Fanuc TP program (LS listing): message22.ls

/PROG  MESSAGE22	  Macro
/ATTR
OWNER		= MNEDITOR;
COMMENT		= "USER MESSAGE";
PROG_SIZE	= 279;
CREATE		= DATE 22-05-23  TIME 16:17:10;
MODIFIED	= DATE 22-05-23  TIME 16:26:38;
FILE_NAME	= MESSAGE2;
VERSION		= 0;
LINE_COUNT	= 3;
MEMORY_SIZE	= 655;
PROTECT		= READ_WRITE;
TCD:  STACK_SIZE	= 0,
      TASK_PRIORITY	= 50,
      TIME_SLICE	= 0,
      BUSY_LAMP_OFF	= 0,
      ABORT_REQUEST	= 0,
      PAUSE_REQUEST	= 7;
DEFAULT_GROUP	= *,*,*,*,*;
CONTROL_CODE	= 00000000 00000000;
/APPL
/APPL

AUTO_SINGULARITY_HEADER;
  ENABLE_SINGULARITY_AVOIDANCE   : FALSE;
/MN
   1:  CALL MESSAGE20    ;
   2:  CALL FAULT_MESSAGE('TP estop pressed.') ;
   3:   ;
/POS
/END
